{attribute 'qualified_only'}
{attribute 'strict'}
{attribute 'to_string'}
TYPE E_DemoStep :
(
	Init := 0,
	WaitForSwitch,
	DetectMovers,
	SortMovers,	
	Enabling,
	SquareUpMovers,
	MoveToSeqenceStartPos,
	JoinTrack,
	FigureEight,
	LeaveTrack,
	GoToOpositeCorner,
	FlyBy,
	MoveAroundPerimeter,
	MoveToCenterOfTiles,
	RotateInverse,
	Spin,
	Lift,
	Tilt,
	Disable,
	//added for ADLM
	ADLM_Step1, // L_move for test tubes AND RotateInverse for Pipeting
	ADLM_Step2, // traverse to start positions for Gripper AND dispensing head
	ADLM_Step3, // cycle through six tubes AND start Pipeting sequence
	ADLM_Step4, // Spin Test tubes AND finish Pipeting sequence
	ManualMode // basically a do nothing to interact with MC3 Motion UI Mover View.
);
END_TYPE

(* stored: Version 1.1.0.1, ProductVersion 3.1.4026.19
   DUT E_DemoStep: Id {ec2e79b1-db13-496a-827a-4cb926db1174} *)
